FUNCTION_BLOCK TestSimple (* Example for a Simple Function Block Type *)
  (* Standard: 61499-1 *)
  (* Version 1.0, 2023-11-29, franz *)
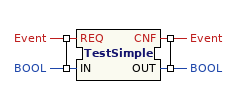
  EVENT_INPUT
    REQ WITH IN; (* Normal Execution Request *)
  END_EVENT
  EVENT_OUTPUT
    CNF WITH OUT; (* Execution Confirmation *)
  END_EVENT
  VAR_INPUT
    IN : BOOL; (* Input *)
  END_VAR
  VAR_OUTPUT
    OUT : BOOL; (* Output *)
  END_VAR
  ALGORITHM REQ IN ST:
OUT := IN;
  END_ALGORITHM
END_FUNCTION_BLOCK
